Fanuc KAREL source: MOVE_FILE.kl

PROGRAM T
%NOLOCKGROUP
VAR
 v0 : STRING[40]
 v1 : INTEGER
BEGIN
 MOVE_FILE(v0, v1)
END T
